Yaskawa INFORM job: JLTV_FENDERS.JBI

/JOB
//NAME JLTV_FENDERS
//POS
///NPOS 269,0,0,0,0,0
///TOOL 0
///POSTYPE PULSE
///PULSE
C00000=-63956,-155140,126844,-105312,-81594,-126671
C00001=2277,-175097,-2251,-89130,-118675,-145962
C00002=2277,-175097,-73511,-89130,-118675,-145962
C00003=-14919,-145236,-96932,-70203,-62356,-69910
C00004=-12571,-128354,-81958,-69802,-60541,-69547
C00005=-9693,-128327,-81950,-68556,-58812,-69965
C00006=-9776,-130540,-82055,-67985,-59270,-70600
C00007=-9648,-130961,-82069,-67809,-59276,-70744
C00008=-8821,-131366,-83195,-68766,-57933,-69654
C00009=20753,-133504,-83242,-50449,-42247,-77185
C00010=38395,-132602,-83224,-34642,-34338,-84273
C00011=38395,-132602,-83224,-34642,-34338,-84273
C00012=38395,-132602,-83224,-34642,-34338,-84273
C00013=46540,-132344,-83219,-25216,-31650,-88760
C00014=62271,-134725,-84753,-3523,-29599,-99395
C00015=62271,-134725,-84753,-3523,-29599,-99395
C00016=62271,-134725,-84753,-3523,-29599,-99395
C00017=126744,-141761,-85039,44788,-42718,-121783
C00018=170872,-134518,-86161,63635,-51905,-130721
C00019=170872,-134518,-86161,63635,-51905,-130721
C00020=170872,-134518,-86161,63635,-51905,-130721
C00021=173979,-137075,-86702,49076,-41409,-124440
C00022=177565,-141459,-86593,28939,-35628,-114869
C00023=177565,-141459,-86593,28939,-35628,-114869
C00024=177565,-141459,-86593,28939,-35628,-114869
C00025=184395,-141855,-86584,36484,-38257,-118288
C00026=207288,-145185,-86329,45569,-44354,-121830
C00027=215126,-147422,-86082,40789,-43387,-119516
C00028=234760,-149730,-85758,24573,-39409,-112238
C00029=235666,-149498,-85796,25700,-39536,-112755
C00030=231834,-148274,-87933,23935,-35240,-110085
C00031=232655,-145301,-86199,25279,-34843,-110781
C00032=233490,-143326,-86367,26956,-34075,-111698
C00033=235167,-141590,-86475,29578,-33725,-113041
C00034=239901,-137156,-86591,36862,-33374,-116796
C00035=239901,-137156,-86591,36862,-33374,-116796
C00036=239468,-136162,-86588,36855,-32802,-116883
C00037=237629,-135533,-86580,35068,-31861,-116098
C00038=237628,-135533,-86580,35068,-31861,-116097
C00039=237628,-135533,-86580,35068,-31861,-116097
C00040=218182,-136250,-86797,8311,-27475,-103121
C00041=199000,-135790,-86962,-20944,-28517,-88743
C00042=179349,-133927,-87055,-45277,-34599,-77018
C00043=159611,-130626,-86983,-62111,-43909,-69236
C00044=145529,-127158,-86730,-70768,-51669,-65334
C00045=130467,-122247,-86132,-77875,-60661,-62089
C00046=83194,-113064,-83981,-83056,-68438,-59002
C00047=78693,-112529,-83889,-83202,-68392,-58892
C00048=74489,-111789,-83746,-83334,-68233,-58745
C00049=73544,-111588,-83705,-83363,-68179,-58706
C00050=71095,-111953,-83785,-82570,-66015,-58963
C00051=70316,-112049,-83805,-82301,-65294,-59047
C00052=64607,-108335,-82945,-84172,-68993,-57875
C00053=64607,-108335,-82945,-84172,-68993,-57875
C00054=64136,-107505,-82741,-84388,-69280,-57667
C00055=64180,-106814,-82564,-84480,-69220,-57512
C00056=65353,-102298,-81335,-84934,-68243,-56551
C00057=65365,-101792,-81187,-85006,-68216,-56439
C00058=65096,-101209,-81016,-85135,-68383,-56302
C00059=63609,-100005,-80655,-85543,-69375,-55994
C00060=65076,-98279,-80119,-85558,-68305,-55681
C00061=65076,-104011,-94976,-87379,-67998,-53005
C00062=220717,-141041,-90238,11451,-28453,-4789
C00063=220975,-137121,-84638,11538,-29263,-4789
C00064=220975,-137121,-84638,11538,-29263,-4789
C00065=220717,-141041,-90238,11451,-28453,-4789
C00066=199102,-139407,-88796,9590,-28908,-4543
C00067=199120,-136374,-84475,9440,-29513,-4446
C00068=199120,-136374,-84475,9440,-29513,-4446
C00069=199083,-141898,-92281,9708,-28445,-4620
C00070=178923,-138415,-89506,13633,-27643,-6713
C00071=178917,-135935,-85869,13376,-28176,-6557
C00072=178918,-135934,-85867,13376,-28174,-6558
C00073=178929,-140078,-91911,13801,-27302,-6816
C00074=136784,-136135,-90977,12891,-25633,-6309
C00075=136821,-131901,-84550,12478,-26662,-6049
C00076=136821,-131901,-84550,12478,-26662,-6049
C00077=136784,-136135,-90977,12891,-25633,-6309
C00078=116236,-133182,-89154,12589,-24985,-5878
C00079=116351,-129669,-83692,12351,-25914,-5713
C00080=116351,-129669,-83692,12351,-25914,-5713
C00081=116236,-133182,-89154,12589,-24985,-5878
C00082=99776,-128761,-86950,16980,-25758,-8059
C00083=99873,-125474,-81794,16601,-26637,-7809
C00084=99873,-125474,-81794,16601,-26637,-7809
C00085=99776,-128761,-86950,16980,-25758,-8059
C00086=-102104,-119076,-89909,9234,-19016,-4103
C00087=-101846,-113640,-80223,8871,-21083,-3859
C00088=-101846,-113640,-80223,8871,-21083,-3859
C00089=-102103,-119074,-89907,9234,-19016,-4101
C00090=-117140,-120986,-88380,10075,-18589,-4492
C00091=-116984,-118182,-83286,9853,-19706,-4344
C00092=-116984,-118182,-83286,9853,-19706,-4344
C00093=-117140,-120986,-88380,10075,-18589,-4492
C00094=-131755,-124810,-89915,20409,-21092,-10530
C00095=-131755,-121478,-84153,19399,-22200,-9932
C00096=-131755,-121478,-84153,19399,-22200,-9932
C00097=-131755,-124810,-89915,20409,-21092,-10530
C00098=-167467,-132124,-89619,18924,-25728,-9507
C00099=-167483,-128719,-84338,18313,-26578,-9138
C00100=-167483,-128719,-84338,18313,-26578,-9138
C00101=-167467,-132124,-89619,18924,-25728,-9507
C00102=-185587,-135717,-88967,20910,-28804,-10331
C00103=-185631,-131903,-83354,20310,-29595,-9962
C00104=-185631,-131903,-83354,20310,-29595,-9962
C00105=-185587,-135717,-88967,20910,-28804,-10331
C00106=-204786,-140151,-90113,23051,-30728,-11203
C00107=-204840,-135592,-83651,22405,-31544,-10800
C00108=-204840,-135592,-83651,22405,-31544,-10800
C00109=-204786,-140151,-90113,23051,-30728,-11203
C00110=-98882,-108096,-90687,24490,-12786,85255
C00111=-98967,-103416,-80523,20155,-15259,87251
C00112=-97852,-105630,-81028,21768,-16361,86433
C00113=-99680,-106251,-81246,17130,-16141,88913
C00114=-100198,-106592,-81344,15734,-16161,89661
C00115=-100511,-107148,-81484,14768,-16308,90184
C00116=-100975,-111608,-82438,12292,-18002,91556
C00117=-101540,-112709,-82663,10744,-18368,92387
C00118=-102184,-112972,-82732,9260,-18389,93172
C00119=-102184,-112972,-82732,9260,-18389,93172
C00120=-102184,-112972,-82732,9260,-18389,93172
C00121=-108013,-114780,-82925,5472,-19155,95226
C00122=-116840,-116513,-83068,-265,-19997,98303
C00123=-146733,-120960,-83565,-18317,-23379,107824
C00124=-216927,-136801,-86187,12872,-29907,93134
C00125=-216927,-136801,-86187,12872,-29907,93134
C00126=-216927,-136801,-86187,12872,-29907,93134
C00127=-218997,-137809,-86138,9794,-30181,94660
C00128=-218163,-138925,-86064,10765,-30877,94218
C00129=-201250,-139768,-85931,41252,-38690,80123
C00130=-201238,-140170,-86483,41322,-38642,80077
C00131=-198492,-141344,-86649,43380,-40171,79283
C00132=-197185,-141944,-86581,44244,-40976,78989
C00133=-193532,-144082,-87766,46896,-42930,77981
C00134=-189225,-145903,-87504,49451,-45599,77216
C00135=-161176,-140691,-87718,53943,-45352,74220
C00136=-139359,-130450,-87301,61141,-45159,69438
C00137=-139359,-130450,-87301,61141,-45159,69438
C00138=-139359,-130450,-87301,61141,-45159,69438
C00139=-132912,-127574,-86938,58041,-40392,71241
C00140=-113538,-124299,-86526,69909,-51239,65867
C00141=-113538,-124299,-86526,69909,-51239,65867
C00142=-113538,-124299,-86526,69909,-51239,65867
C00143=-75200,-125420,-86004,71442,-54907,65170
C00144=-63437,-122754,-85604,73468,-55667,64524
C00145=-51827,-118403,-84555,74560,-55830,64078
C00146=-51827,-118403,-84555,74560,-55830,64078
C00147=-51827,-118403,-84555,74560,-55830,64078
C00148=-45819,-116324,-84253,77094,-59520,62836
C00149=-38911,-115626,-84093,79241,-64029,62049
C00150=-38911,-115626,-84093,79241,-64029,62049
C00151=-38911,-115626,-84093,79241,-64029,62049
C00152=-34206,-127012,-86472,69078,-50186,67076
C00153=-23646,-133800,-86712,59791,-45202,71681
C00154=-23646,-133800,-86712,59791,-45202,71681
C00155=-23646,-133800,-86712,59791,-45202,71681
C00156=-22723,-133554,-86712,60473,-45648,71368
C00157=-22017,-133082,-86712,61106,-45922,71033
C00158=-20875,-130784,-86594,62743,-46037,70003
C00159=-20215,-128094,-84987,63617,-46156,69457
C00160=-18086,-122552,-84408,66988,-46344,67228
C00161=-18086,-133952,-103979,70615,-44891,64381
C00162=1141,-175007,-98783,66988,-102227,67229
C00163=1141,-175089,26483,66988,-118571,67229
C00164=-171943,-158203,65342,62007,-93837,-40952
C00165=-174843,-156250,61168,59943,-92878,-47560
C00166=-174884,-149197,69874,59946,-93261,-47211
C00167=-174236,-145812,71072,59372,-79857,-47597
C00168=-172797,-142378,72122,59705,-67414,-47916
C00169=-172723,-139545,76281,59522,-67720,-47588
C00170=-173073,-136776,80369,59088,-68118,-47294
C00171=-172602,-136370,80359,57471,-61055,-46594
C00172=-171863,-135569,80782,55633,-54067,-45714
C00173=-170756,-134112,81941,53010,-46264,-44367
C00174=-169588,-132253,83740,49922,-39669,-42716
C00175=-172202,-124939,97020,46177,-42296,-35162
C00176=-175201,-116137,112510,42585,-45408,-27548
C00177=-179725,-103865,133025,38625,-49589,-17846
C00178=-182437,-114887,111199,33836,-41135,-14978
C00179=-185919,-121262,97597,22370,-34375,-7559
C00180=-189325,-123826,91203,7367,-32006,1988
C00181=-192934,-128813,83866,6501,-30996,977
C00182=-194297,-129800,82349,6130,-30775,628
C00183=-195986,-128931,83114,5622,-30748,223
C00184=-200133,-125525,84758,9437,-30950,-748
C00185=-212327,-118926,93911,3550,-38568,-2588
C00186=-227854,-119648,90309,-2688,-37161,-1056
C00187=-232068,-133509,73423,-4245,-32198,2480
C00188=-224801,-145212,56791,-38949,-36183,24271
C00189=-219295,-151149,49486,-53357,-50276,34921
C00190=-216154,-154041,46440,-57718,-63792,39342
C00191=-214471,-155816,44737,-59342,-76359,41874
C00192=-212181,-163317,32818,-63987,-82994,54441
C00193=-210239,-167534,24858,-63389,-87774,62652
C00194=-209501,-170544,20161,-62902,-87471,63069
C00195=-214511,-173113,26018,-66265,-88769,60803
C00196=-183241,-141368,78763,-57333,-96573,-54831
C00197=-181431,-143869,70974,-55878,-95500,-53479
C00198=-181431,-143869,70974,-55878,-95500,-53479
C00199=-183241,-141368,78763,-57333,-96573,-54831
C00200=-185236,-123918,103372,-57487,-90922,-57084
C00201=-183217,-128516,91143,-56174,-89322,-55173
C00202=-183217,-128516,91143,-56174,-89322,-55173
C00203=-185236,-123918,103372,-57487,-90922,-57084
C00204=-127582,-141773,109706,-82308,-91591,-67971
C00205=-132307,-145418,62418,-85570,-87578,-56085
C00206=-131977,-148633,51964,-85512,-87333,-54105
C00207=-131977,-148633,51964,-85512,-87333,-54105
C00208=-132307,-145418,62418,-85570,-87578,-56085
C00209=-132116,-116858,103710,-85204,-88156,-59409
C00210=-131789,-122725,88363,-85163,-87809,-56827
C00211=-131789,-122725,88363,-85163,-87809,-56827
C00212=-132116,-116858,103710,-85204,-88156,-59409
C00213=-132086,-175086,28776,-85496,-87491,-55195
C00214=167780,-151019,89189,-65646,-98497,-64716
C00215=163256,-141921,95136,-50992,-75767,-63693
C00216=164622,-146954,83379,-50923,-74033,-62057
C00217=164622,-146954,83379,-50923,-74033,-62057
C00218=163256,-141921,95136,-50992,-75767,-63693
C00219=159916,-125941,115697,-44667,-63049,-66644
C00220=161601,-134840,95747,-45983,-59633,-63954
C00221=161601,-134840,95747,-45983,-59633,-63954
C00222=159112,-118425,131428,-43671,-65725,-68501
C00223=216933,-125941,115697,-73773,-63049,-66644
C00224=214319,-150024,53932,-92267,-59650,-53288
C00225=214024,-151691,47364,-93906,-59717,-51729
C00226=214024,-151691,47364,-93906,-59717,-51729
C00227=214319,-150024,53932,-92267,-59650,-53288
C00228=212765,-167272,33315,-94222,-59464,-52337
C00229=212278,-169046,25414,-96366,-59658,-50384
C00230=212278,-169046,25414,-96366,-59658,-50384
C00231=212765,-167272,33315,-94222,-59464,-52337
C00232=204018,-163525,44974,-122210,86547,-147941
C00233=199154,-168652,34335,-129636,87230,-149952
C00234=199154,-158927,45235,-129654,87525,-149752
C00235=198806,-153563,50444,-127783,87206,-155518
C00236=198006,-159000,41811,-126294,86795,-161513
C00237=197336,-163523,33608,-124896,86563,-167364
C00238=197738,-163257,33757,-124610,86484,-167375
C00239=197980,-162795,34403,-124448,86509,-167327
C00240=201825,-143194,68341,-122020,89699,-154997
C00241=201823,-130263,85945,-120968,76208,-144776
C00242=202996,-116534,106328,-127689,66571,-134239
C00243=206954,-124935,89202,-136006,48218,-130911
C00244=210457,-127584,83786,-143959,39184,-126357
C00245=218557,-129412,78540,-175081,27944,-108392
C00246=206826,-126980,85258,-178941,30212,-110975
C00247=189127,-120496,100790,-183813,34613,-105483
C00248=187506,-122818,100198,-184163,35485,-105961
C00249=186226,-123679,99777,-184469,35694,-106318
C00250=184567,-121660,103508,-184812,36495,-106815
C00251=180993,-112256,119434,-185366,39559,-108020
C00252=174981,-117693,112007,-190403,32708,-106439
C00253=169780,-119924,110312,-195278,27866,-104575
C00254=166131,-117722,116190,-194529,29417,-99161
C00255=164787,-117304,117471,-194360,29750,-97171
C00256=160549,-119668,113510,-194686,28720,-90661
C00257=155581,-123216,107082,-195282,27004,-82901
C00258=158627,-126564,104239,-214214,37078,-72930
C00259=160614,-126632,105782,-222278,46686,-69184
C00260=161923,-125473,108710,-226824,54765,-67543
C00261=163089,-122938,113719,-231055,64100,-66608
C00262=164497,-135614,96784,-234283,68690,-64762
C00263=165745,-147161,82855,-237100,74663,-63560
C00264=165227,-147668,81665,-237480,74337,-63452
C00265=163066,-136963,105784,-237298,77357,-66819
C00266=51354,-175100,27099,-75814,-41400,-97395
C00267=-14969,-152284,67590,-92780,-64518,-114234
C00268=-63956,-155140,126844,-105312,-81594,-126671
//INST
///DATE 2022/10/06 11:32
///ATTR SC,RW
///GROUP1 RB1
NOP
MOVJ C00000 VJ=65.00  //HOME
CALL JOB:SYS_GATE_LOCK
CALL JOB:SYS_VERIFY_GATE_LOCKED
CALL JOB:SYS_SPINDLE_START
CALL JOB:SYS_FILTERS_START
MOVJ C00001 VJ=65.00
MOVJ C00002 VJ=65.00
MOVJ C00003 VJ=65.00  //ABOVE LEFT FRONT
MOVL C00004 V=15.0  //INTO LEFT TOP
MOVL C00005 V=15.0  //UP TO EDGE
MOVL C00006 V=15.0  //INSIDE CORNER
MOVL C00007 V=15.0
MOVC C00008 V=15.0
MOVC C00009 V=15.0
MOVC C00010 V=15.0
MOVL C00011 V=15.0
MOVC C00012 V=15.0
MOVC C00013 V=15.0
MOVC C00014 V=15.0
MOVL C00015 V=15.0
MOVC C00016 V=15.0
MOVC C00017 V=15.0
MOVC C00018 V=15.0
MOVL C00019 V=15.0
MOVC C00020 V=15.0
MOVC C00021 V=15.0
MOVC C00022 V=15.0
MOVL C00023 V=15.0
MOVC C00024 V=15.0
MOVC C00025 V=15.0
MOVC C00026 V=15.0
MOVC C00027 V=15.0
MOVC C00028 V=15.0
MOVL C00029 V=15.0
MOVL C00030 V=15.0
MOVC C00031 V=15.0
MOVC C00032 V=15.0
MOVC C00033 V=15.0
MOVL C00034 V=15.0
MOVC C00035 V=15.0
MOVC C00036 V=15.0
MOVC C00037 V=15.0
MOVL C00038 V=15.0
MOVC C00039 V=15.0  //START OUTSIDE CURVE
MOVC C00040 V=15.0
MOVC C00041 V=15.0
MOVC C00042 V=15.0
MOVC C00043 V=15.0
MOVC C00044 V=15.0
MOVC C00045 V=15.0
MOVC C00046 V=15.0
MOVC C00047 V=15.0
MOVC C00048 V=15.0
MOVC C00049 V=15.0
MOVC C00050 V=15.0
MOVC C00051 V=15.0
MOVL C00052 V=15.0
MOVC C00053 V=15.0
MOVC C00054 V=15.0
MOVC C00055 V=15.0
MOVL C00056 V=15.0
MOVL C00057 V=15.0
MOVL C00058 V=15.0
MOVL C00059 V=15.0
MOVL C00060 V=15.0  //OUT
MOVJ C00061 VJ=65.00  //ABOVE
MOVJ C00062 VJ=65.00  //ABOVE 1ST -375
MOVL C00063 V=15.0  //INTO .375
FORMCUT FCF#(5)
MOVL C00064 V=15.0
FORMCUT FCF#(5)
MOVJ C00065 VJ=25.00  //OUT
MOVJ C00066 VJ=65.00  //ABOVE 2ND
MOVL C00067 V=15.0  //INTO
FORMCUT FCF#(5)
MOVL C00068 V=15.0
FORMCUT FCF#(5)
MOVJ C00069 VJ=25.00 PL=8  //OUT
MOVJ C00070 VJ=65.00  //ABOVE 3RD
MOVL C00071 V=15.0  //INTO
FORMCUT FCF#(5)
MOVL C00072 V=15.0
FORMCUT FCF#(5)
MOVJ C00073 VJ=25.00 PL=8  //OUT
MOVJ C00074 VJ=65.00  //ABOVE 4TH
MOVL C00075 V=15.0  //INTO
FORMCUT FCF#(5)
MOVL C00076 V=15.0
FORMCUT FCF#(5)
MOVJ C00077 VJ=25.00 PL=8  //OUT
MOVJ C00078 VJ=65.00  //ABOVE 5TH
MOVL C00079 V=15.0  //INTO
FORMCUT FCF#(5)
MOVL C00080 V=15.0
FORMCUT FCF#(5)
MOVJ C00081 VJ=25.00 PL=8  //OUT
MOVJ C00082 VJ=65.00  //ABOVE 6TH
MOVL C00083 V=15.0  //INTO
FORMCUT FCF#(5)
MOVL C00084 V=15.0
FORMCUT FCF#(5)
MOVJ C00085 VJ=25.00 PL=8  //OUT
MOVJ C00086 VJ=65.00  //ABOVE 1ST
MOVL C00087 V=15.0  //INTO
FORMCUT FCF#(5)
MOVL C00088 V=15.0
FORMCUT FCF#(5)
MOVJ C00089 VJ=25.00  //OUT
MOVJ C00090 VJ=65.00  //ABOVE 2ND
MOVL C00091 V=15.0  //INTO
FORMCUT FCF#(5)
MOVL C00092 V=15.0
FORMCUT FCF#(5)
MOVJ C00093 VJ=25.00 PL=8  //OUT
MOVJ C00094 VJ=65.00  //ABOVE 3RD
MOVL C00095 V=15.0  //INTO
FORMCUT FCF#(5)
MOVL C00096 V=15.0
FORMCUT FCF#(5)
MOVJ C00097 VJ=25.00 PL=8  //OUT
MOVJ C00098 VJ=65.00  //ABOVE 4TH
MOVL C00099 V=15.0
FORMCUT FCF#(5)
MOVL C00100 V=15.0
FORMCUT FCF#(5)
MOVJ C00101 VJ=25.00 PL=8  //OUT
MOVJ C00102 VJ=65.00  //ABOVE 5TH
MOVL C00103 V=15.0  //INTO
FORMCUT FCF#(5)
MOVL C00104 V=15.0
FORMCUT FCF#(5)
MOVJ C00105 VJ=25.00 PL=8  //OUT
MOVJ C00106 VJ=65.00  //ABOVE 6TH
MOVL C00107 V=15.0  //INTO
FORMCUT FCF#(5)
MOVL C00108 V=15.0
FORMCUT FCF#(5)
MOVJ C00109 VJ=25.00 PL=8  //OUT
MOVJ C00110 VJ=65.00  //ROTATE
MOVL C00111 V=150.0  //UP TO PART
MOVL C00112 V=15.0  //CORNER
MOVL C00113 V=15.0
MOVL C00114 V=15.0
MOVL C00115 V=15.0
MOVC C00116 V=15.0
MOVC C00117 V=15.0
MOVC C00118 V=15.0
MOVL C00119 V=15.0
MOVC C00120 V=15.0
MOVC C00121 V=15.0
MOVC C00122 V=15.0
MOVC C00123 V=15.0
MOVC C00124 V=15.0
MOVL C00125 V=15.0
MOVC C00126 V=15.0
MOVC C00127 V=15.0
MOVC C00128 V=15.0
MOVL C00129 V=15.0
MOVC C00130 V=15.0
MOVC C00131 V=15.0
MOVC C00132 V=15.0
MOVL C00133 V=15.0
MOVC C00134 V=15.0  //START INSIDE CURVE
MOVC C00135 V=15.0
MOVC C00136 V=15.0
MOVL C00137 V=15.0
MOVC C00138 V=15.0
MOVC C00139 V=15.0
MOVC C00140 V=15.0
MOVL C00141 V=15.0
MOVC C00142 V=15.0
MOVC C00143 V=15.0
MOVC C00144 V=15.0
MOVC C00145 V=15.0
MOVL C00146 V=15.0
MOVC C00147 V=15.0
MOVC C00148 V=15.0
MOVC C00149 V=15.0
MOVL C00150 V=15.0
MOVC C00151 V=15.0
MOVC C00152 V=15.0
MOVC C00153 V=15.0
MOVL C00154 V=15.0
MOVC C00155 V=15.0
MOVC C00156 V=15.0
MOVC C00157 V=15.0
MOVL C00158 V=15.0
MOVL C00159 V=15.0
MOVL C00160 V=15.0  //OUT
MOVJ C00161 VJ=65.00  //ABOVE
MOVJ C00162 VJ=65.00
MOVJ C00163 VJ=65.00  //OUTSIDE
MOVJ C00164 VJ=65.00  //LEFT SIDE
MOVL C00165 V=150.0  //ABOVE PART
MOVL C00166 V=15.0  //INTO PART
MOVL C00167 V=15.0
MOVC C00168 V=15.0
MOVC C00169 V=15.0
MOVC C00170 V=15.0
MOVL C00171 V=15.0
MOVL C00172 V=15.0
MOVL C00173 V=15.0
MOVL C00174 V=15.0
MOVL C00175 V=15.0
MOVL C00176 V=15.0
MOVL C00177 V=15.0
MOVL C00178 V=15.0
MOVL C00179 V=15.0
MOVL C00180 V=15.0
MOVC C00181 V=15.0
MOVC C00182 V=15.0
MOVC C00183 V=15.0
MOVL C00184 V=15.0
MOVL C00185 V=15.0
MOVL C00186 V=15.0
MOVL C00187 V=15.0
MOVL C00188 V=15.0
MOVL C00189 V=15.0
MOVL C00190 V=15.0
MOVL C00191 V=15.0
MOVL C00192 V=15.0
MOVL C00193 V=15.0
MOVL C00194 V=15.0  //END
MOVJ C00195 VJ=25.00  //AWAY
MOVJ C00196 VJ=65.00  //UP TO TOP HOLE
MOVL C00197 V=15.0  //INTO TOP FRONT
FORMCUT FCF#(5)
MOVL C00198 V=15.0
FORMCUT FCF#(5)
MOVJ C00199 VJ=25.00 PL=8
MOVJ C00200 VJ=65.00  //UP TO
MOVL C00201 V=15.0  //INTO BOTTOM HOLE
FORMCUT FCF#(5)
MOVL C00202 V=15.0
FORMCUT FCF#(5)
MOVJ C00203 VJ=25.00 PL=8  //OUT
MOVJ C00204 VJ=65.00  //LEFT SIDE
MOVJ C00205 VJ=65.00  //UP TO
MOVL C00206 V=15.0  //INTO TOP SIDE HOLE
FORMCUT FCF#(5)
MOVL C00207 V=15.0
FORMCUT FCF#(5)
MOVJ C00208 VJ=25.00 PL=8  //OUT OF
MOVJ C00209 VJ=65.00  //UP TO
MOVL C00210 V=15.0  //INTO BOTTOM SIDE
FORMCUT FCF#(5)
MOVL C00211 V=15.0
FORMCUT FCF#(5)
MOVJ C00212 VJ=25.00 PL=8  //OUT OF
MOVJ C00213 VJ=65.00  //READY
MOVJ C00214 VJ=65.00  //RIGHT SIDE
MOVJ C00215 VJ=65.00  //UP TO
MOVL C00216 V=15.0  //INTO TOP HOLE
FORMCUT FCF#(5)
MOVL C00217 V=15.0
FORMCUT FCF#(5)
MOVJ C00218 VJ=25.00 PL=8  //OUT OF
MOVJ C00219 VJ=65.00  //UP TO
MOVL C00220 V=15.0  //INTO BOTTOM HOLE
FORMCUT FCF#(5)
MOVL C00221 V=15.0
FORMCUT FCF#(5)
MOVJ C00222 VJ=25.00  //OUT OF
MOVJ C00223 VJ=65.00
MOVJ C00224 VJ=65.00  //UP TO BOTTOM HOLE
MOVL C00225 V=15.0  //INTO
FORMCUT FCF#(5)
MOVL C00226 V=15.0
FORMCUT FCF#(5)
MOVJ C00227 VJ=25.00 PL=8  //OUT OF BOTTOM HOLE
MOVJ C00228 VJ=65.00  //UP TO TOP HOLE
MOVL C00229 V=15.0  //INTO TOP HOLE
FORMCUT FCF#(5)
MOVL C00230 V=15.0
FORMCUT FCF#(5)
MOVJ C00231 VJ=25.00 PL=8  //OUT OF HOLE
MOVJ C00232 VJ=65.00
MOVJ C00233 VJ=65.00
MOVL C00234 V=15.0  //INTO
MOVL C00235 V=15.0
MOVL C00236 V=15.0
MOVL C00237 V=15.0
MOVL C00238 V=15.0
MOVL C00239 V=15.0
MOVL C00240 V=15.0
MOVL C00241 V=15.0
MOVL C00242 V=15.0
MOVL C00243 V=15.0
MOVL C00244 V=15.0
MOVL C00245 V=15.0
MOVL C00246 V=15.0  //BOTTOM
MOVL C00247 V=15.0
MOVC C00248 V=15.0
MOVC C00249 V=15.0
MOVC C00250 V=15.0
MOVL C00251 V=15.0
MOVL C00252 V=15.0
MOVL C00253 V=15.0
MOVL C00254 V=15.0
MOVL C00255 V=15.0
MOVL C00256 V=15.0
MOVL C00257 V=15.0
MOVL C00258 V=15.0
MOVL C00259 V=15.0
MOVL C00260 V=15.0
MOVL C00261 V=15.0  //POINT
MOVL C00262 V=15.0
MOVL C00263 V=15.0  //END
MOVJ C00264 VJ=65.00  //AWAY
MOVJ C00265 VJ=65.00  //OUT
MOVJ C00266 VJ=65.00
MOVJ C00267 VJ=65.00
MOVJ C00268 VJ=65.00  //HOME
CALL JOB:SYS_SPINDLE_STOP
CALL JOB:SYS_FILTERS_STOP
CALL JOB:SYS_UNLOCK_GATE
END
